INTERFACE I_DatatypePack

METHOD RegisterWith
VAR_INPUT
	Datatypes : I_Datatypes;
END_VAR
END_METHOD

END_INTERFACE

(* stored: Version 1.1.0.1, ProductVersion 3.1.4024.12
   Itf I_DatatypePack: Id {494942d1-e598-081b-32e2-4b26f595758c}
   Method RegisterWith: Id {008c9af1-6678-02e0-2f3d-79bc95210dc2} *)
